Staubli VAL3: write_to_file.pgx

program write_to_file(num x_nX (dimensions=1), num x_nY (dimensions=1), string x_sItem (dimensions=1), bool x_bCall (dimensions=1))
  local num i
  local num l_nSize
  local string l_sFill
begin
  //
  // check the size
  //
  l_nSize=size(sWrite)-x_nY
  if l_nSize<=0
    for i=0 to abs(l_nSize)
      // insert new Line
      insert(sWrite[size(sWrite)])
    endFor
  endIf
  //
  // write in the line
  //
  // test if the len is ok
  //
  l_nSize=len(sWrite[x_nY])-x_nX
  if l_nSize<=0
    for i=0 to abs(l_nSize)
      // insert white space if the item on the left is a PROG
      sWrite[x_nY]=insert(sWrite[x_nY]," ",len(sWrite[x_nY]))
    endFor
    // insert the line
    sWrite[x_nY]=replace(sWrite[x_nY],x_sItem,0,x_nX)
  else
    if x_bCall
      //need to insert for all the line an empty string of nChar
      for i=0 to size(sWrite)-1
        call use:strfill(l_sFill,nChar+1,l_sFill)
        //        if (mid(sWrite[i],1,x_nX+nChar)=="═")
        //          call use:strfillchr(l_sFill,l_sFill,"═")
        //          // line
        //          sWrite[i]=insert(sWrite[i],l_sFill,x_nX+nChar+1)
        //        else
        // space
        sWrite[i]=insert(sWrite[i],l_sFill,x_nX+nChar+1)
        //       endIf
      endFor
    endIf
    // replace the string
    sWrite[x_nY]=replace(sWrite[x_nY],x_sItem,nChar+1,x_nX)
  endIf
end
